FUNCTION_BLOCK TEST_START_FB
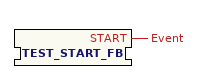
  EVENT_OUTPUT
    START;
  END_EVENT
  EC_STATES
    START;
  END_STATES
END_FUNCTION_BLOCK
